Staubli VAL3: pallet_resetAll.pgx

program pallet_resetAll()
begin
  // resetAll the pallet
  call pallet_resetAll()
end
